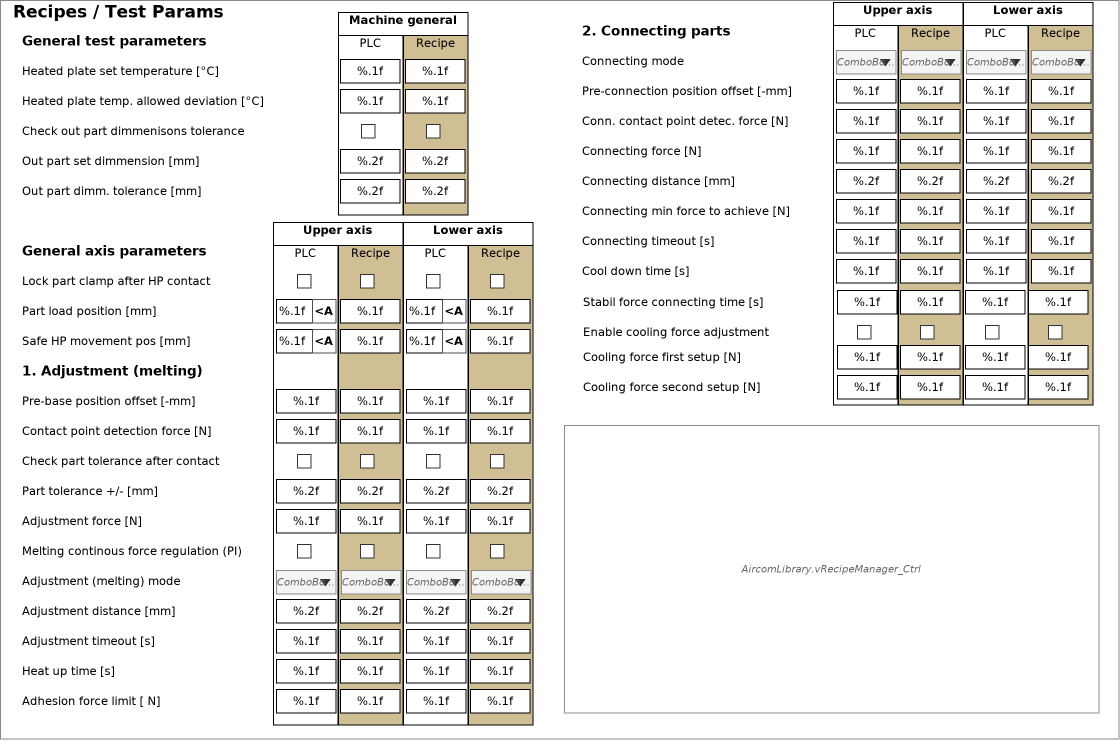
VISUALIZATION vHP3_MachineSub_TestParams  // 1120x740
VAR_IN_OUT
	fbHP: fbHPv3_Control;
//	stParams: stHPv3_TestParams;
//	stRecipe: stHPv3_TestParams;
END_VAR
    RoundedRectangle (273,222 130x503), "Upper axis"
    RoundedRectangle (273,245 65x480), "PLC"
    RoundedRectangle (338,245 65x480), "Recipe"
    RoundedRectangle (403,222 130x503), "Lower axis"
    RoundedRectangle (468,245 65x480), "Recipe"
    RoundedRectangle (403,245 65x480), "PLC"
    Label (19,239 260x24), "General axis parameters"
    Label (19,269 230x24), "Lock part clamp after HP contact"
    Checkbox (295,269 24x24), variable: fbHP.stTestData.stAxisUp_Data.bPartLockAfterHpContact
    Checkbox (358,269 24x24), variable: fbHP.stTmpRecipeData.stAxisUp_Data.bPartLockAfterHpContact
    Checkbox (424,269 24x24), variable: fbHP.stTestData.stAxisDn_Data.bPartLockAfterHpContact
    Checkbox (488,269 24x24), variable: fbHP.stTmpRecipeData.stAxisDn_Data.bPartLockAfterHpContact
    Label (19,299 230x24), "Part load position [mm]"
    Rectangle (276,299 60x24), "%.1f", text variable: fbHP.stTestData.stAxisUp_Data.lrPartLoadPosition_mm
        OnMouseDown: write the text variable via Default, min 20, max 200, title 'Part load position', format %.1f
    Rectangle (340,299 60x24), "%.1f", text variable: fbHP.stTmpRecipeData.stAxisUp_Data.lrPartLoadPosition_mm
        OnMouseDown: write the text variable via Default, min 20, max 200, title 'Part load position', format %.1f
    Rectangle (406,299 60x24), "%.1f", text variable: fbHP.stTestData.stAxisDn_Data.lrPartLoadPosition_mm
        OnMouseDown: write the text variable via Default, min 20, max 200, title 'Part load position', format %.1f
    Rectangle (470,299 60x24), "%.1f", text variable: fbHP.stTmpRecipeData.stAxisDn_Data.lrPartLoadPosition_mm
        OnMouseDown: write the text variable via Default, min 20, max 200, title 'Part load position', format %.1f
    Label (19,329 230x24), "Safe HP movement pos [mm]"
    Rectangle (276,329 60x24), "%.1f", text variable: fbHP.stTestData.stAxisUp_Data.lrSafeHpMovementPos_mm
        OnMouseDown: write the text variable via Default, min 5, max 200, title 'Safe HP movement pos', format %.1f
    Rectangle (340,329 60x24), "%.1f", text variable: fbHP.stTmpRecipeData.stAxisUp_Data.lrSafeHpMovementPos_mm
        OnMouseDown: write the text variable via Default, min 5, max 200, title 'Safe HP movement pos', format %.1f
    Rectangle (406,329 60x24), "%.1f", text variable: fbHP.stTestData.stAxisDn_Data.lrSafeHpMovementPos_mm
        OnMouseDown: write the text variable via Default, min 5, max 200, title 'Safe HP movement pos', format %.1f
    Rectangle (470,329 60x24), "%.1f", text variable: fbHP.stTmpRecipeData.stAxisDn_Data.lrSafeHpMovementPos_mm
        OnMouseDown: write the text variable via Default, min 5, max 200, title 'Safe HP movement pos', format %.1f
    Label (19,359 260x24), "1. Adjustment (melting)"
    Label (19,569 230x24), "Adjustment (melting) mode"
    ComboBoxInteger (276,570 60x24), variable: fbHP.stTestData.stAxisUp_Data.nMeltingMode
    ComboBoxInteger (341,570 60x24), variable: fbHP.stTmpRecipeData.stAxisUp_Data.nMeltingMode
    ComboBoxInteger (406,570 60x24), variable: fbHP.stTestData.stAxisDn_Data.nMeltingMode
    ComboBoxInteger (471,570 60x24), variable: fbHP.stTmpRecipeData.stAxisDn_Data.nMeltingMode
    Label (19,539 230x24), "Melting continous force regulation (PI)"
    Checkbox (295,539 24x24), variable: fbHP.stTestData.stAxisUp_Data.bMeltingForceRegulation
    Checkbox (358,539 24x24), variable: fbHP.stTmpRecipeData.stAxisUp_Data.bMeltingForceRegulation
    Checkbox (424,539 24x24), variable: fbHP.stTestData.stAxisDn_Data.bMeltingForceRegulation
    Checkbox (488,539 24x24), variable: fbHP.stTmpRecipeData.stAxisDn_Data.bMeltingForceRegulation
    Label (19,509 230x24), "Adjustment force [N]"
    Rectangle (276,509 60x24), "%.1f", text variable: fbHP.stTestData.stAxisUp_Data.rMeltingForce_N
        OnMouseDown: write the text variable via Default, min 10, max 200, title 'Adjustment max force', format %.1f
    Rectangle (340,509 60x24), "%.1f", text variable: fbHP.stTmpRecipeData.stAxisUp_Data.rMeltingForce_N
        OnMouseDown: write the text variable via Default, min 10, max 200, title 'Adjustment max force', format %.1f
    Rectangle (406,509 60x24), "%.1f", text variable: fbHP.stTestData.stAxisDn_Data.rMeltingForce_N
        OnMouseDown: write the text variable via Default, min 10, max 200, title 'Adjustment max force', format %.1f
    Rectangle (470,509 60x24), "%.1f", text variable: fbHP.stTmpRecipeData.stAxisDn_Data.rMeltingForce_N
        OnMouseDown: write the text variable via Default, min 10, max 200, title 'Adjustment max force', format %.1f
    Label (19,599 230x24), "Adjustment distance [mm]"
    Rectangle (276,599 60x24), "%.2f", text variable: fbHP.stTestData.stAxisUp_Data.lrMeltingDistance_mm
        OnMouseDown: write the text variable via Default, min 0.01, max 200, title 'Melting distance', format %.2f
    Rectangle (340,599 60x24), "%.2f", text variable: fbHP.stTmpRecipeData.stAxisUp_Data.lrMeltingDistance_mm
        OnMouseDown: write the text variable via Default, min 0.01, max 200, title 'Melting distance', format %.2f
    Rectangle (406,599 60x24), "%.2f", text variable: fbHP.stTestData.stAxisDn_Data.lrMeltingDistance_mm
        OnMouseDown: write the text variable via Default, min 0.01, max 200, title 'Melting distance', format %.2f
    Rectangle (470,599 60x24), "%.2f", text variable: fbHP.stTmpRecipeData.stAxisDn_Data.lrMeltingDistance_mm
        OnMouseDown: write the text variable via Default, min 0.01, max 200, title 'Melting distance', format %.2f
    Label (19,389 230x24), "Pre-base position offset [-mm]"
    Rectangle (276,389 60x24), "%.1f", text variable: fbHP.stTestData.stAxisUp_Data.lrPreBaseOffset_mm
        OnMouseDown: write the text variable via Default, min 0.5, max 10, title 'Pre-base position offset', format %.1f
    Rectangle (340,389 60x24), "%.1f", text variable: fbHP.stTmpRecipeData.stAxisUp_Data.lrPreBaseOffset_mm
        OnMouseDown: write the text variable via Default, min 0.5, max 10, title 'Pre-base position offset', format %.1f
    Rectangle (406,389 60x24), "%.1f", text variable: fbHP.stTestData.stAxisDn_Data.lrPreBaseOffset_mm
        OnMouseDown: write the text variable via Default, min 0.5, max 10, title 'Pre-base position offset', format %.1f
    Rectangle (470,389 60x24), "%.1f", text variable: fbHP.stTmpRecipeData.stAxisDn_Data.lrPreBaseOffset_mm
        OnMouseDown: write the text variable via Default, min 0.5, max 10, title 'Pre-base position offset', format %.1f
    Label (19,629 230x24), "Adjustment timeout [s]"
    Rectangle (276,629 60x24), "%.1f", text variable: fbHP.stTestData.stAxisUp_Data.rMeltingTimeout_s
        OnMouseDown: write the text variable via Default, min 2, max 30, title 'Adjustment timeout [s]', format %.1f
    Rectangle (340,629 60x24), "%.1f", text variable: fbHP.stTmpRecipeData.stAxisUp_Data.rMeltingTimeout_s
        OnMouseDown: write the text variable via Default, min 2, max 30, title 'Adjustment timeout [s]', format %.1f
    Rectangle (406,629 60x24), "%.1f", text variable: fbHP.stTestData.stAxisDn_Data.rMeltingTimeout_s
        OnMouseDown: write the text variable via Default, min 2, max 30, title 'Adjustment timeout [s]', format %.1f
    Rectangle (470,629 60x24), "%.1f", text variable: fbHP.stTmpRecipeData.stAxisDn_Data.rMeltingTimeout_s
        OnMouseDown: write the text variable via Default, min 2, max 30, title 'Adjustment timeout [s]', format %.1f
    Label (19,419 230x24), "Contact point detection force [N]"
    Rectangle (276,419 60x24), "%.1f", text variable: fbHP.stTestData.stAxisUp_Data.rAdjContactDetectForce_N
        OnMouseDown: write the text variable via Default, min 2, max 40, title 'Contact detection force', format %.1f
    Rectangle (340,419 60x24), "%.1f", text variable: fbHP.stTmpRecipeData.stAxisUp_Data.rAdjContactDetectForce_N
        OnMouseDown: write the text variable via Default, min 2, max 40, title 'Contact detection force', format %.1f
    Rectangle (406,419 60x24), "%.1f", text variable: fbHP.stTestData.stAxisDn_Data.rAdjContactDetectForce_N
        OnMouseDown: write the text variable via Default, min 2, max 40, title 'Contact detection force', format %.1f
    Rectangle (470,419 60x24), "%.1f", text variable: fbHP.stTmpRecipeData.stAxisDn_Data.rAdjContactDetectForce_N
        OnMouseDown: write the text variable via Default, min 2, max 40, title 'Contact detection force', format %.1f
    RoundedRectangle (833,2 130x293), "Upper axis"
    RoundedRectangle (833,25 65x380), "PLC"
    RoundedRectangle (898,25 65x380), "Recipe"
    RoundedRectangle (963,2 130x293), "Lower axis"
    RoundedRectangle (1028,25 65x380), "Recipe"
    RoundedRectangle (963,25 65x380), "PLC"
    Label (19,689 230x24), "Adhesion force limit [ N]"
    Rectangle (276,689 60x24), "%.1f", text variable: fbHP.stTestData.stAxisUp_Data.rAdhesionForceLimit_N
        OnMouseDown: write the text variable via Default, min 0, max 100, title 'Adhesion force limit', format %.1f
    Rectangle (340,689 60x24), "%.1f", text variable: fbHP.stTmpRecipeData.stAxisUp_Data.rAdhesionForceLimit_N
        OnMouseDown: write the text variable via Default, min 0, max 100, title 'Adhesion force limit', format %.1f
    Rectangle (406,689 60x24), "%.1f", text variable: fbHP.stTestData.stAxisDn_Data.rAdhesionForceLimit_N
        OnMouseDown: write the text variable via Default, min 0, max 100, title 'Adhesion force limit', format %.1f
    Rectangle (470,689 60x24), "%.1f", text variable: fbHP.stTmpRecipeData.stAxisDn_Data.rAdhesionForceLimit_N
        OnMouseDown: write the text variable via Default, min 0, max 100, title 'Adhesion force limit', format %.1f
    Label (579,49 230x24), "Connecting mode"
    Label (579,139 230x24), "Connecting force [N]"
    Label (579,259 230x24), "Cool down time [s]"
    Label (579,169 230x24), "Connecting distance [mm]"
    Label (579,79 230x24), "Pre-connection position offset [-mm]"
    Label (579,229 230x24), "Connecting timeout [s]"
    Label (579,109 230x24), "Conn. contact point detec. force [N]"
    Label (579,19 260x24), "2. Connecting parts"
    Label (579,199 230x24), "Connecting min force to achieve [N]"
    Label (19,29 260x24), "General test parameters"
    RoundedRectangle (338,12 130x203), "Machine general"
    RoundedRectangle (338,35 65x180), "PLC"
    RoundedRectangle (403,35 65x180), "Recipe"
    Label (19,59 300x24), "Heated plate set temperature [°C]"
    Rectangle (340,59 60x24), "%.1f", text variable: fbHP.stTestData.rHeatedPlateSetTemperature
        OnMouseDown: write the text variable via Default, min 150, max 300, title 'Heated plate temperature', format %.1f
    Rectangle (405,59 60x24), "%.1f", text variable: fbHP.stTmpRecipeData.rHeatedPlateSetTemperature
        OnMouseDown: write the text variable via Default, min 150, max 300, title 'Heated plate temperature', format %.1f
    Label (19,89 300x24), "Heated plate temp. allowed deviation [°C]"
    Rectangle (340,89 60x24), "%.1f", text variable: fbHP.stTestData.rHeatedPlateAllowDeviation
        OnMouseDown: write the text variable via Default, min 3, max 30, title 'Heated plate temp. deviation', format %.1f
    Rectangle (405,89 60x24), "%.1f", text variable: fbHP.stTmpRecipeData.rHeatedPlateAllowDeviation
        OnMouseDown: write the text variable via Default, min 3, max 30, title 'Heated plate temp. deviation', format %.1f
    Label (19,119 300x24), "Check out part dimmenisons tolerance"
    Checkbox (359,119 24x24), variable: fbHP.stTestData.bCheckOutPartDimmension_EN
    Checkbox (424,119 24x24), variable: fbHP.stTmpRecipeData.bCheckOutPartDimmension_EN
    Label (19,149 300x24), "Out part set dimmension [mm]"
    Rectangle (340,149 60x24), "%.2f", text variable: fbHP.stTestData.lrOutPartDesiredDimm_mm
        OnMouseDown: write the text variable via Default, min 10, max 200, title 'Out part height', format %.2f
    Rectangle (405,149 60x24), "%.2f", text variable: fbHP.stTmpRecipeData.lrOutPartDesiredDimm_mm
        OnMouseDown: write the text variable via Default, min 10, max 200, title 'Out part height', format %.2f
    Label (19,179 300x24), "Out part dimm. tolerance [mm]"
    Rectangle (340,179 60x24), "%.2f", text variable: fbHP.stTestData.lrOutPartDimmTolerance_mm
        OnMouseDown: write the text variable via Default, min 0.02, max 10, title 'Out part height tolerance', format %.2f
    Rectangle (405,179 60x24), "%.2f", text variable: fbHP.stTmpRecipeData.lrOutPartDimmTolerance_mm
        OnMouseDown: write the text variable via Default, min 0.02, max 10, title 'Out part height tolerance', format %.2f
    Label (19,449 230x24), "Check part tolerance after contact"
    Checkbox (295,449 24x24), variable: fbHP.stTestData.stAxisUp_Data.bCheckPartToleranceAfterContact
    Checkbox (358,449 24x24), variable: fbHP.stTmpRecipeData.stAxisUp_Data.bCheckPartToleranceAfterContact
    Checkbox (424,449 24x24), variable: fbHP.stTestData.stAxisDn_Data.bCheckPartToleranceAfterContact
    Checkbox (488,449 24x24), variable: fbHP.stTmpRecipeData.stAxisDn_Data.bCheckPartToleranceAfterContact
    Label (19,479 230x24), "Part tolerance +/- [mm]"
    Rectangle (276,479 60x24), "%.2f", text variable: fbHP.stTestData.stAxisUp_Data.lrPartToleranceFromBasePos_mm
        OnMouseDown: write the text variable via Default, min 0.01, max 10, title 'Part tolerance', format %.2f
    Rectangle (340,479 60x24), "%.2f", text variable: fbHP.stTmpRecipeData.stAxisUp_Data.lrPartToleranceFromBasePos_mm
        OnMouseDown: write the text variable via Default, min 0.01, max 10, title 'Part tolerance', format %.2f
    Rectangle (406,479 60x24), "%.2f", text variable: fbHP.stTestData.stAxisDn_Data.lrPartToleranceFromBasePos_mm
        OnMouseDown: write the text variable via Default, min 0.01, max 10, title 'Part tolerance', format %.2f
    Rectangle (470,479 60x24), "%.2f", text variable: fbHP.stTmpRecipeData.stAxisDn_Data.lrPartToleranceFromBasePos_mm
        OnMouseDown: write the text variable via Default, min 0.01, max 10.0, title 'Part tolerance', format %.2f
    Label (19,659 230x24), "Heat up time [s]"
    Rectangle (276,659 60x24), "%.1f", text variable: fbHP.stTestData.stAxisUp_Data.rHeatingUpTime_s
        OnMouseDown: write the text variable via Default, min 2, max 60, title 'Heat up time [s]', format %.1f
    Rectangle (340,659 60x24), "%.1f", text variable: fbHP.stTmpRecipeData.stAxisUp_Data.rHeatingUpTime_s
        OnMouseDown: write the text variable via Default, min 2, max 60, title 'Heat up time [s]', format %.1f
    Rectangle (406,659 60x24), "%.1f", text variable: fbHP.stTestData.stAxisDn_Data.rHeatingUpTime_s
        OnMouseDown: write the text variable via Default, min 2, max 60, title 'Heat up time [s]', format %.1f
    Rectangle (470,659 60x24), "%.1f", text variable: fbHP.stTmpRecipeData.stAxisDn_Data.rHeatingUpTime_s
        OnMouseDown: write the text variable via Default, min 2, max 60, title 'Heat up time [s]', format %.1f
    Frame (564,425 535x288)
        shows AircomLibrary.vRecipeManager_Ctrl(fbRecipe := fbHP.fbRecipes)
    Rectangle (312,299 24x24), "<A"
        OnMouseClick: execute { fbHP.stTestData.stAxisUp_Data.lrPartLoadPosition_mm := fbHP.fbAxisUp.ActualPosition; }
    Rectangle (312,329 24x24), "<A"
        OnMouseClick: execute { fbHP.stTestData.stAxisUp_Data.lrSafeHpMovementPos_mm := fbHP.fbAxisUp.ActualPosition; }
    Rectangle (442,329 24x24), "<A"
        OnMouseClick: execute { fbHP.stTestData.stAxisDn_Data.lrSafeHpMovementPos_mm := fbHP.fbAxisDn.ActualPosition; }
    Rectangle (442,299 24x24), "<A"
        OnMouseClick: execute { fbHP.stTestData.stAxisDn_Data.lrPartLoadPosition_mm := fbHP.fbAxisDn.ActualPosition; }
    RoundedRectangle (10,0 300x26), "Recipes / Test Params"
    Label (580,375 230x24), "Cooling force second setup [N]"
    Label (580,345 230x24), "Cooling force first setup [N]"
    Label (580,290 230x24), "Stabil force connecting time [s]"
    Group (836,50 61x349), input disabled if: TRUE
        ComboBoxInteger (0,0 60x24), variable: fbHP.stTestData.stAxisUp_Data.nConnectingMode
        Rectangle (0,89 60x24), "%.1f", text variable: fbHP.stTestData.stAxisUp_Data.rConnectingForce_N
            OnMouseDown: write the text variable via Default, min 5, max 100, title 'Connecting max force', format %.1f
        Rectangle (0,209 60x24), "%.1f", text variable: fbHP.stTestData.stAxisUp_Data.rCoolingDownTime_s
            OnMouseDown: write the text variable via Default, min 2, max 60, title 'Cool down time [s]', format %.1f
        Rectangle (0,119 60x24), "%.2f", text variable: fbHP.stTestData.stAxisUp_Data.lrConnectingDistance_mm
            OnMouseDown: write the text variable via Default, min 0.02, max 200, title 'Connectiong distance', format %.2f
        Rectangle (0,29 60x24), "%.1f", text variable: fbHP.stTestData.stAxisUp_Data.lrPreConnectingOffset_mm
            OnMouseDown: write the text variable via Default, min 0.5, max 10, title 'Pre-connection position offset', format %.1f
        Rectangle (0,179 60x24), "%.1f", text variable: fbHP.stTestData.stAxisUp_Data.rConnectingTimeout_s
            OnMouseDown: write the text variable via Default, min 2, max 30, title 'Connecting timeout [s]', format %.1f
        Rectangle (0,59 60x24), "%.1f", text variable: fbHP.stTestData.stAxisUp_Data.rConContactDetecForce_N
            OnMouseDown: write the text variable via Default, min 2, max 40, title 'Connecting contact detection force', format %.1f
        Rectangle (0,149 60x24), "%.1f", text variable: fbHP.stTestData.stAxisUp_Data.rConnectingMinForce_N
            OnMouseDown: write the text variable via Default, min 2, max 100, title 'Connecting min force to achieve', format %.1f
        Rectangle (1,325 60x24), "%.1f", text variable: fbHP.stTestData.stAxisUp_Data.rSecondCoolingforceSetUp
            OnMouseDown: write the text variable via Default, min 2, max 60, title 'Cool down time [s]', format %.1f
        Rectangle (1,295 60x24), "%.1f", text variable: fbHP.stTestData.stAxisUp_Data.rFirstCoolingForceSetUp
            OnMouseDown: write the text variable via Default, min 2, max 60, title 'Cool down time [s]', format %.1f
        Rectangle (1,240 60x24), "%.1f", text variable: fbHP.stTestData.stAxisUp_Data.rStabilForceConnectingTime
            OnMouseDown: write the text variable via Default, min 2, max 60, title 'Cool down time [s]', format %.1f
        Checkbox (19,270 24x24), variable: fbHP.stTestData.stAxisUp_Data.bAllowCoolingForceAquire
    Label (580,320 230x24), "Enable cooling force adjustment"
    Group (900,50 61x349), input disabled if: TRUE
        ComboBoxInteger (1,0 60x24), variable: fbHP.stTmpRecipeData.stAxisUp_Data.nConnectingMode
        Rectangle (0,89 60x24), "%.1f", text variable: fbHP.stTmpRecipeData.stAxisUp_Data.rConnectingForce_N
            OnMouseDown: write the text variable via Default, min 5, max 100, title 'Connecting max force', format %.1f
        Rectangle (0,209 60x24), "%.1f", text variable: fbHP.stTmpRecipeData.stAxisUp_Data.rCoolingDownTime_s
            OnMouseDown: write the text variable via Default, min 2, max 60, title 'Cool down time [s]', format %.1f
        Rectangle (0,119 60x24), "%.2f", text variable: fbHP.stTmpRecipeData.stAxisUp_Data.lrConnectingDistance_mm
            OnMouseDown: write the text variable via Edit, min 0.02, max 200, title 'Connectiong distance', format %.2f
        Rectangle (0,29 60x24), "%.1f", text variable: fbHP.stTmpRecipeData.stAxisUp_Data.lrPreConnectingOffset_mm
            OnMouseDown: write the text variable via Default, min 0.5, max 10, title 'Pre-connection position offset', format %.1f
        Rectangle (0,179 60x24), "%.1f", text variable: fbHP.stTmpRecipeData.stAxisUp_Data.rConnectingTimeout_s
            OnMouseDown: write the text variable via Default, min 2, max 30, title 'Connecting timeout [s]', format %.1f
        Rectangle (0,59 60x24), "%.1f", text variable: fbHP.stTmpRecipeData.stAxisUp_Data.rConContactDetecForce_N
            OnMouseDown: write the text variable via Default, min 2, max 40, title 'Connecting contact detection force', format %.1f
        Rectangle (0,149 60x24), "%.1f", text variable: fbHP.stTmpRecipeData.stAxisUp_Data.rConnectingMinForce_N
            OnMouseDown: write the text variable via Default, min 2, max 100, title 'Connecting min force to achieve', format %.1f
        Rectangle (0,240 60x24), "%.1f", text variable: fbHP.stTmpRecipeData.stAxisUp_Data.rStabilForceConnectingTime
            OnMouseDown: write the text variable via Default, min 2, max 60, title 'Cool down time [s]', format %.1f
        Rectangle (0,325 60x24), "%.1f", text variable: fbHP.stTmpRecipeData.stAxisUp_Data.rSecondCoolingforceSetUp
            OnMouseDown: write the text variable via Default, min 2, max 60, title 'Cool down time [s]', format %.1f
        Rectangle (0,295 60x24), "%.1f", text variable: fbHP.stTmpRecipeData.stAxisUp_Data.rFirstCoolingForceSetUp
            OnMouseDown: write the text variable via Default, min 2, max 60, title 'Cool down time [s]', format %.1f
        Checkbox (18,270 24x24), variable: fbHP.stTmpRecipeData.stAxisUp_Data.bAllowCoolingForceAquire
    Group (965,50 61x349)
        ComboBoxInteger (1,0 60x24), variable: fbHP.stTestData.stAxisDn_Data.nConnectingMode
        Rectangle (1,89 60x24), "%.1f", text variable: fbHP.stTestData.stAxisDn_Data.rConnectingForce_N
            OnMouseDown: write the text variable via Default, min 5, max 100, title 'Connecting max force', format %.1f
        Rectangle (1,209 60x24), "%.1f", text variable: fbHP.stTestData.stAxisDn_Data.rCoolingDownTime_s
            OnMouseDown: write the text variable via Default, min 2, max 60, title 'Cool down time [s]', format %.1f
        Rectangle (1,119 60x24), "%.2f", text variable: fbHP.stTestData.stAxisDn_Data.lrConnectingDistance_mm
            OnMouseDown: write the text variable via Default, min 0.02, max 200, title 'Connectiong distance', format %.2f
        Rectangle (1,29 60x24), "%.1f", text variable: fbHP.stTestData.stAxisDn_Data.lrPreConnectingOffset_mm
            OnMouseDown: write the text variable via Default, min 0.5, max 10, title 'Pre-connection position offset', format %.1f
        Rectangle (1,179 60x24), "%.1f", text variable: fbHP.stTestData.stAxisDn_Data.rConnectingTimeout_s
            OnMouseDown: write the text variable via Default, min 2, max 30, title 'Connecting timeout [s]', format %.1f
        Rectangle (1,59 60x24), "%.1f", text variable: fbHP.stTestData.stAxisDn_Data.rConContactDetecForce_N
            OnMouseDown: write the text variable via Default, min 2, max 40, title 'Connecting contact detection force', format %.1f
        Rectangle (1,149 60x24), "%.1f", text variable: fbHP.stTestData.stAxisDn_Data.rConnectingMinForce_N
            OnMouseDown: write the text variable via Default, min 2, max 100, title 'Connecting min force to achieve', format %.1f
        Rectangle (0,240 60x24), "%.1f", text variable: fbHP.stTestData.stAxisDn_Data.rStabilForceConnectingTime
            OnMouseDown: write the text variable via Default, min 2, max 60, title 'Cool down time [s]', format %.1f
        Rectangle (0,325 60x24), "%.1f", text variable: fbHP.stTestData.stAxisDn_Data.rSecondCoolingforceSetUp
            OnMouseDown: write the text variable via Default, min 2, max 60, title 'Cool down time [s]', format %.1f
        Rectangle (0,295 60x24), "%.1f", text variable: fbHP.stTestData.stAxisDn_Data.rFirstCoolingForceSetUp
            OnMouseDown: write the text variable via Default, min 2, max 60, title 'Cool down time [s]', format %.1f
        Checkbox (18,270 24x24), variable: fbHP.stTestData.stAxisDn_Data.bAllowCoolingForceAquire
    Group (1028,50 63x349)
        ComboBoxInteger (3,0 60x24), variable: fbHP.stTmpRecipeData.stAxisDn_Data.nConnectingMode
        Rectangle (3,89 60x24), "%.1f", text variable: fbHP.stTmpRecipeData.stAxisDn_Data.rConnectingForce_N
            OnMouseDown: write the text variable via Default, min 5, max 100, title 'Connecting max force', format %.1f
        Rectangle (3,209 60x24), "%.1f", text variable: fbHP.stTmpRecipeData.stAxisDn_Data.rCoolingDownTime_s
            OnMouseDown: write the text variable via Default, min 2, max 60, title 'Cool down time [s]', format %.1f
        Rectangle (3,119 60x24), "%.2f", text variable: fbHP.stTmpRecipeData.stAxisDn_Data.lrConnectingDistance_mm
            OnMouseDown: write the text variable via Default, min 0.02, max 200, title 'Connectiong distance', format %.2f
        Rectangle (3,29 60x24), "%.1f", text variable: fbHP.stTmpRecipeData.stAxisDn_Data.lrPreConnectingOffset_mm
            OnMouseDown: write the text variable via Default, min 0.5, max 10, title 'Pre-connection position offset', format %.1f
        Rectangle (3,179 60x24), "%.1f", text variable: fbHP.stTmpRecipeData.stAxisDn_Data.rConnectingTimeout_s
            OnMouseDown: write the text variable via Default, min 2, max 30, title 'Connecting timeout [s]', format %.1f
        Rectangle (3,59 60x24), "%.1f", text variable: fbHP.stTmpRecipeData.stAxisDn_Data.rConContactDetecForce_N
            OnMouseDown: write the text variable via Default, min 2, max 40, title 'Connecting contact detection force', format %.1f
        Rectangle (3,149 60x24), "%.1f", text variable: fbHP.stTmpRecipeData.stAxisDn_Data.rConnectingMinForce_N
            OnMouseDown: write the text variable via Default, min 2, max 100, title 'Connecting min force to achieve', format %.1f
        Rectangle (0,240 60x24), "%.1f", text variable: fbHP.stTmpRecipeData.stAxisUp_Data.rStabilForceConnectingTime
            OnMouseDown: write the text variable via Default, min 2, max 60, title 'Cool down time [s]', format %.1f
        Rectangle (0,325 60x24), "%.1f", text variable: fbHP.stTmpRecipeData.stAxisDn_Data.rSecondCoolingforceSetUp
            OnMouseDown: write the text variable via Default, min 2, max 60, title 'Cool down time [s]', format %.1f
        Rectangle (0,295 60x24), "%.1f", text variable: fbHP.stTmpRecipeData.stAxisDn_Data.rFirstCoolingForceSetUp
            OnMouseDown: write the text variable via Default, min 2, max 60, title 'Cool down time [s]', format %.1f
        Checkbox (18,270 24x24), variable: fbHP.stTmpRecipeData.stAxisDn_Data.bAllowCoolingForceAquire
END_VISUALIZATION

(* stored: Version 1.1.0.1, ProductVersion 3.1.4024.15
   Visu vHP3_MachineSub_TestParams: Id {fac2a841-e321-44dc-bd76-de45893aab59} *)
